****Commands (Commands are identified by an '.' located at the first byte in the command string):
".THIS.XXXXXX;" Will allow access to variables in the current communication object. (since the client don't know which to connection object in the array it's connected to ) 
example:
".THIS.stSettings.nADSPORT=852;" will change the default ADS-port to 852.  .THIS will simply replace  the path to the communication object with the correct connection index (x):
".THIS.stSettings.nADSPORT=852;" = "Main.fbServer.aApplications[x].stSettings.nADSPORT=852;"
example 2:
".THIS.stSettings.nConnectionIndex?;" will retrun the connection index for the current connection. 


".ADR.IDXGRP,IDXOFF,size,adst_type;". The ADR command allows reading and writing to variables with absoulte adress
example: Access softlimits of axis 1 in motion (NC). Adresses can be find in documentation on by hovering over the parameter in NC (tool tip) or by right clicking on the parameter of intrest and choosing properties. NC has ADSPort 501 
Writing: "ADSPORT=501/.ADR.16#5001,16#D,8,5=-100;" 
Reading: "ADSPORT=501/.ADR.16#5001,16#D,8,5?;"
Note: Axis 2 can be accessed in the same way by increasing the IDXGRP to 5002  (axis 3=> 5003)
 
example 2: Reading the absoute adress of an variable with symbolic adress

"ADSPORT=852/.ADR.Main.sVersion?; Will return the absolute adress of the variable Main.sVersion at ADS-port 852.

*)

END_PROGRAM

// ---- POUs/Static Command support/FB_GetStaticADR.TcPOU
FUNCTION_BLOCK FB_GetStaticADR
VAR
	sVersion: STRING:='0.9.0';
END_VAR
VAR_INPUT
	bEnable:BOOL:=FALSE;
	nCommadStartIndex:INT:=0;
	nCommandEndIndex:INT:=0;	
END_VAR
VAR
	psCommandBufferString: POINTER TO STRING; //string to point into byte buffer	
	nQuestionSign: INT;
END_VAR

VAR_IN_OUT
	byteCommandBuffer	:	ARRAY[0..PLCPRJ_BUFFER_SIZE] OF BYTE;//ADS input buffer
	nBytesInCommandBuffer:DINT:=0;
	nIndexEndOfCommand:DINT:=0;
END_VAR

VAR_OUTPUT
	nErrorId: UDINT;
	bError:BOOL:=FALSE;
	sVariableName:STRING(255);
	sSubErrorString: STRING;
END_VAR

//Static command/option 1: Check if ADR option	
(*IF bEnable THEN
	bError:=FALSE;
	nErrorId:=0;	
	sSubErrorString:='';	
	sVariableName:='';		
	psCommandBufferString:=ADR(byteCommandBuffer);
	nQuestionSign:=len(STR:=EPICS_STATIC_COMMAND_ABS_ADRESS);
	IF 	byteCommandBuffer[len(STR:=EPICS_STATIC_COMMAND_ABS_ADRESS)]=EPICS_ASCII_QUESTIONMARK AND nQuestionSign>0 THEN
		sVariableName:=right(str:=left(str:=PSTRING_TO_STRING(psCommandBufferString),size:=nCommandEndIndex-1),SIZE:=(nCommandEndIndex-1)-nQuestionSign-1);
		IF NOT F_RemoveBytesFromBuffer_V1_00(nRemoveBytes:= nCommandEndIndex,byteCommandBuffer:=byteCommandBuffer,nBytesInCommandBuffer:=nBytesInCommandBuffer,nIndexEndOfCommand:=nIndexEndOfCommand) THEN 			
			bError:=TRUE;
			nErrorId:=312;
			sSubErrorString:='State 3: Failed to clear buffer (ADR).';	
		END_IF
	ELSE
		nErrorId:=313;
		bError:=TRUE;
		sSubErrorString:='State 3: Failed to parse ADR set command.';	
	END_IF		
END_IF*)

END_FUNCTION_BLOCK

// ---- POUs/Static Command support/FB_ParseStaticCommand.TcPOU
FUNCTION_BLOCK FB_ParseStaticCommand
VAR
	sVersion: STRING:='0.9.0';
END_VAR
VAR
	psCommandBufferString: POINTER TO STRING; //string to point into byte buffer		
	nEqualSign: INT;
	nQuestionMark: INT;
END_VAR

VAR_IN_OUT
	byteCommandBuffer	:	ARRAY[0..PLCPRJ_BUFFER_SIZE] OF BYTE;//ADS input buffer
	nBytesInCommandBuffer:DINT:=0;
	nIndexEndOfCommand:DINT:=0;
END_VAR

VAR_OUTPUT
	nErrorId: UDINT;
	bError:BOOL:=FALSE;
	sSubErrorString: STRING;
	sStaticCommand:STRING;
	sStaticValue:STRING;
	bReadCommand:BOOL:=FALSE;
	bWriteCommand:BOOL:=FALSE;
END_VAR

//Parse static command	
nErrorId:=0;
bError:=FALSE;
sStaticCommand:='';
sStaticValue:='';
bReadCommand:=FALSE;
bWriteCommand:=FALSE;
psCommandBufferString:=ADR(byteCommandBuffer);

nEqualSign:=find(STR1:=PSTRING_TO_STRING(psCommandBufferString),STR2:=EPICS_WRITE_CMD);	
IF nEqualSign>0 AND nEqualSign<=nIndexEndOfCommand THEN
	bWriteCommand:=TRUE;	
	//Command
	memcpy(destAddr:=ADR(sStaticCommand[0]),srcAddr:=ADR(byteCommandBuffer[0]),n:=nEqualSign-1);
	memset(destAddr	:=ADR(sStaticCommand[nEqualSign-1]),fillByte:=0,n:=1);				//Terminate string	
	//Value
	memcpy(destAddr:=ADR(sStaticValue[0]),srcAddr:=ADR(byteCommandBuffer[nEqualSign]),n:=nIndexEndOfCommand-nEqualSign-1);
	memset(destAddr	:=ADR(sStaticValue[nIndexEndOfCommand-nEqualSign-1]),fillByte:=0,n:=1); //Terminate string
	IF NOT F_RemoveBytesFromBuffer_V1_00(nRemoveBytes:= nIndexEndOfCommand,byteCommandBuffer:=byteCommandBuffer,nBytesInCommandBuffer:=nBytesInCommandBuffer,nIndexEndOfCommand:=nIndexEndOfCommand) THEN 			
		bError:=TRUE;
		nErrorId:=301;
		sSubErrorString:='State 3: Failed to clear buffer (Parse static command write).';	
	END_IF				
ELSE
	nQuestionMark:=find(STR1:=PSTRING_TO_STRING(psCommandBufferString),STR2:=EPICS_READ_CMD);	
	IF nQuestionMark>0 AND nQuestionMark<=nIndexEndOfCommand THEN
		bReadCommand:=TRUE;	
		//Command
		memcpy(destAddr:=ADR(sStaticCommand[0]),srcAddr:=ADR(byteCommandBuffer[0]),n:=nQuestionMark-1);
		memset(destAddr	:=ADR(sStaticCommand[nQuestionMark-1]),fillByte:=0,n:=1);				//Terminate string	

		//Clean buffer
		IF NOT F_RemoveBytesFromBuffer_V1_00(nRemoveBytes:= nIndexEndOfCommand,byteCommandBuffer:=byteCommandBuffer,nBytesInCommandBuffer:=nBytesInCommandBuffer,nIndexEndOfCommand:=nIndexEndOfCommand) THEN 			
			bError:=TRUE;
			nErrorId:=302;
			sSubErrorString:='State 3: Failed to clear buffer (Parse static command read).';	
		END_IF		
	END_IF
END_IF	

IF NOT (bReadCommand OR  bWriteCommand) THEN										
	bError:=TRUE;
	nErrorId:=303;
	sSubErrorString:='State 3: Parsing of static command failed.';	
END_IF

END_FUNCTION_BLOCK

// ---- POUs/Static Command support/FB_SetStaticADSPort.TcPOU
FUNCTION_BLOCK FB_SetStaticADSPort
VAR
	sVersion: STRING:='0.9.0';
END_VAR
VAR_INPUT
	bEnable:BOOL:=FALSE;
	nCommadStartIndex:INT:=0;
	nCommandEndIndex:INT:=0;	
END_VAR
VAR
	psCommandBufferString: POINTER TO STRING; //string to point into byte buffer	
	bInStaticSection: BOOL;	
	sTemp: STRING;
	nEqualSign: INT;
END_VAR

VAR_IN_OUT
	byteCommandBuffer	:	ARRAY[0..PLCPRJ_BUFFER_SIZE] OF BYTE;//ADS input buffer
	nBytesInCommandBuffer:DINT:=0;
	nIndexEndOfCommand:DINT:=0;
END_VAR

VAR_OUTPUT
	nErrorId: UDINT;
	bError:BOOL:=FALSE;
	nADSPort: UINT:=0;
	sSubErrorString: STRING;
END_VAR

//Static command/option 1: Check if ADSPORT option	
IF bEnable THEN
	psCommandBufferString:=ADR(byteCommandBuffer);
	nEqualSign:=find(STR1:=PSTRING_TO_STRING(psCommandBufferString),STR2:=EPICS_WRITE_CMD);															
	sTemp:=right(str:=left(str:=PSTRING_TO_STRING(psCommandBufferString),size:=nCommandEndIndex-1),SIZE:=(nCommandEndIndex-1)-nEqualSign);
	nADSPort:=STRING_TO_UINT(sTemp);	
	IF nADSPort<1 OR nADSPort>20000 THEN
		nErrorId:=301;
		bError:=TRUE;
		sSubErrorString:='State 3: ADSPORT out of range.';
	//	nADSPort:=EPICS_ADS_PORT; //Set to default
	END_IF						
	//Remove ADS command from buffer
	IF NOT F_RemoveBytesFromBuffer_V1_00(nRemoveBytes:= nCommandEndIndex,byteCommandBuffer:=byteCommandBuffer,nBytesInCommandBuffer:=nBytesInCommandBuffer,nIndexEndOfCommand:=nIndexEndOfCommand) THEN 			
			bError:=TRUE;
			nErrorId:=302;
			sSubErrorString:='State 3: Failed to clear buffer (ADSPORT)).';	
	END_IF							
END_IF

END_FUNCTION_BLOCK

// ---- POUs/Static Command support/FB_SetStaticADR.TcPOU
FUNCTION_BLOCK FB_SetStaticADR
VAR
	sVersion: STRING:='0.9.0';
END_VAR
VAR_INPUT
	bEnable:BOOL:=FALSE;
	nCommadStartIndex:INT:=0;
	nCommandEndIndex:INT:=0;	
END_VAR
VAR
	psCommandBufferString: POINTER TO STRING; //string to point into byte buffer	
	bInStaticSection: BOOL;	
	sTemp: STRING;
	nEqualSign: INT;
	nComma:INT:=0;
	stemp1: STRING(255);
	sTemp2: STRING(255);
	sTemp3: STRING(255);
	sTemp4: STRING(255);
	sVal:STRING;
	nQuestionSign: INT;
	nRemove: INT;
END_VAR

VAR_IN_OUT
	byteCommandBuffer	:	ARRAY[0..PLCPRJ_BUFFER_SIZE] OF BYTE;//ADS input buffer
	nBytesInCommandBuffer:DINT:=0;
	nIndexEndOfCommand:DINT:=0;
END_VAR

VAR_OUTPUT
	nErrorId: UDINT;
	bError:BOOL:=FALSE;
	stSymInfo:SYMINFOSTRUCT;
	sSubErrorString: STRING;
END_VAR

//Should look like "ADR=idxgrp,idxoff,size,type/"   => ADR=1,2,3,4/
(*
Type:
ADST_BIT             = 33 (&H21)
ADST_INT8            = 16 (&H10)
ADST_INT16           = 2
ADST_INT32           = 3
ADST_INT64           = 20 (&H14)
ADST_UINT8           = 17 (&H11)
ADST_UINT16          = 18 (&H12)
ADST_UINT32          = 19 (&H13)
ADST_UINT64          = 21 (&H15)
ADST_REAL32          = 4
ADST_REAL64          = 5
ADST_REAL80          = 32 (&H20)
ADST_BIGTYPE         = 65 (&H41)
ADST_VOID            = 0
*)

//Static command/option 1: Check if ADR option	
IF bEnable THEN
	bError:=TRUE;
	nErrorId:=0;	
	sSubErrorString:='';	
	stSymInfo.adsDataType:=0;
	stSymInfo.byteSize:=0;
	stSymInfo.idxGroup:=0;
	stSymInfo.idxOffset:=0;
	nRemove:=0;	
	psCommandBufferString:=ADR(byteCommandBuffer);		
	nEqualSign:=find(STR1:=PSTRING_TO_STRING(psCommandBufferString),STR2:=EPICS_WRITE_CMD);															
	sTemp:=right(str:=left(str:=PSTRING_TO_STRING(psCommandBufferString),size:=nCommandEndIndex-1),SIZE:=(nCommandEndIndex)-nEqualSign-1);
	nComma:=find(STR1:=sTemp,STR2:=EPICS_ARRAY_DELIMITER);
	IF 	nComma>0 THEN
		sVal:=left(STR:=sTemp,size:=nComma);
		stSymInfo.idxGroup:=STRING_TO_UDINT(sVal);					
		sTemp1:=right(STR:=sTemp,size:=len(sTemp)-nComma);
		nRemove:=nRemove+nComma+1;		
		nComma:=find(STR1:=sTemp1,STR2:=EPICS_ARRAY_DELIMITER);
		IF 	nComma>0 THEN
			sVal:=left(STR:=sTemp1,size:=nComma);
			stSymInfo.idxOffset:=STRING_TO_UDINT(sVal);					
			sTemp2:=right(STR:=sTemp1,size:=len(sTemp1)-nComma);
			nRemove:=nRemove+nComma+1;
			nComma:=find(STR1:=sTemp2,STR2:=EPICS_ARRAY_DELIMITER); //last			
			IF 	nComma>0 THEN
				sVal:=left(STR:=sTemp2,size:=nComma);
				stSymInfo.byteSize:=STRING_TO_UDINT(sVal);					
				sTemp3:=right(STR:=sTemp2,size:=len(sTemp2)-nComma);		
				nRemove:=nRemove+nComma+1;
				nComma:=len(sTemp3);												
				IF nComma>0 AND find(str1:=stemp3,str2:=EPICS_COMMAND_OPTION_DELIMITER)=0 THEN
					stSymInfo.adsDataType:=STRING_TO_INT(sTemp3);
					nRemove:=nRemove+nComma+1;													
					bError:=FALSE;
				END_IF					
			END_IF							
		END_IF					
	END_IF
	
	IF bError THEN
		nErrorId:=310;
		bError:=TRUE;
		sSubErrorString:='State 3: Failed to parse ADR command.';	
		// try to clean buffers		
		F_RemoveBytesFromBuffer_V1_00(nRemoveBytes:= nRemove,byteCommandBuffer:=byteCommandBuffer,nBytesInCommandBuffer:=nBytesInCommandBuffer,nIndexEndOfCommand:=nIndexEndOfCommand);  		
	ELSE
		IF NOT F_RemoveBytesFromBuffer_V1_00(nRemoveBytes:= nCommandEndIndex,byteCommandBuffer:=byteCommandBuffer,nBytesInCommandBuffer:=nBytesInCommandBuffer,nIndexEndOfCommand:=nIndexEndOfCommand) THEN 			
			bError:=TRUE;
			nErrorId:=311;
			sSubErrorString:='State 3: Failed to clear buffer (ADR).';	
		END_IF	
	END_IF			
END_IF

END_FUNCTION_BLOCK
